// TIA Portal V16 export
// export: Created 2024-12-03T15:41:39.1016418Z, ExportSetting WithDefaults, DisplayName Totally Integrated Automation Portal, DisplayVersion V16 Update 6, DisplayName TIA Portal Version Control Interface, DisplayVersion V16 Update 2, DisplayName TIA Portal Openness, DisplayVersion V16 Update 6, DisplayName TIA Portal Teamcenter Gateway, DisplayVersion V16, DisplayName SINAMICS Startdrive Advanced, DisplayVersion V16 Update 5, DisplayName SINAMICS Startdrive G130, G150, S120, S150, SINAMICS MV, S210, DisplayVersion V16 Update 5, DisplayName SINAMICS Startdrive G110M, G120, G120C, G120D, G120P, G115D, DisplayVersion V16 Update 5, DisplayName STEP 7 Professional, DisplayVersion V16 Update 6, DisplayName STEP 7 Safety, DisplayVersion V16, DisplayName WinCC Advanced / Unified PC, DisplayVersion V16 Update 6
FUNCTION_BLOCK "InputReader_MainRack"   // FB6, SCL
{ S7_Optimized_Access := 'FALSE' }
VERSION : 0.1
// stored: AutoNumber true, IsIECCheckEnabled false, SetENOAutomatically false, UDAEnableTagReadback false
   VAR
      RESET { S7_SetPoint := 'True'} : "SmartBool";
      EMG { S7_SetPoint := 'True'} : "SmartBool";
   END_VAR
   VAR_TEMP
      T_Signal : Bool;
   END_VAR
BEGIN
   REGION RESET SYSTEM

       #T_Signal := "HMI_DB".ResetFromHMI
       OR "ApplicationState_DB".Appstate[0].Hmi_Buttons.reset.SignalFromHMI;

       #RESET(I_Sensor:=#T_Signal,
              HoldOnTIme:=T#0ms,
              O_data=>"Inputs_DB".Reset_System);

        "ApplicationState_DB".Appstate[0].Hmi_Buttons.reset.SignalFromHMI := "ApplicationState_DB".Appstate[0].Hmi_Buttons.reset.SignalFromHMI OR
        "Inputs_DB".Reset_System.LE;

        IF "ApplicationState_DB".Appstate[0].Hmi_Buttons.reset.SignalFromHMI THEN
            "ApplicationState_DB".Appstate[0].Hmi_Buttons.reset.SignalFromHMI := 0;
        END_IF;

   END_REGION

   REGION MAINRACK INPUTS

       #EMG(I_Sensor := "I_EMG_MAIN",
            O_data => "Inputs_DB".EMG_OK);


   END_REGION
END_FUNCTION_BLOCK
